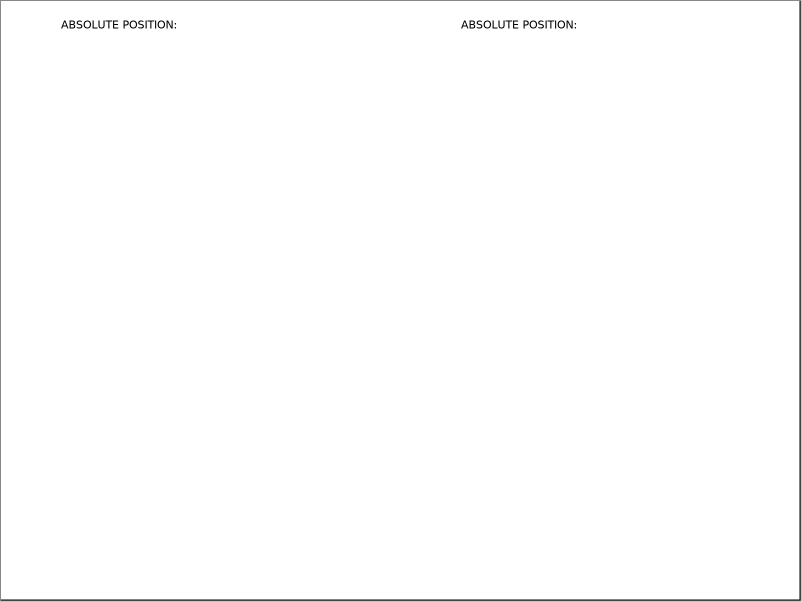
VISUALIZATION F20_Digital_Cam_Switch  // 802x602
    Rectangle (0,0 800x600)
    Label (10,10 170x30), "ABSOLUTE POSITION:"
    Label (410,10 170x30), "ABSOLUTE POSITION:"
END_VISUALIZATION

(* stored: Version 1.1.0.1, ProductVersion 3.1.4022.7
   Visu F20_Digital_Cam_Switch: Id {9a815661-7a31-4313-8ced-4810bbff613b} *)
